FUNCTION_BLOCK FB_Station IMPLEMENTS ITF_Observable
VAR
	//ITF_Observable
	_Observers : ARRAY[1..2] OF ITF_Observer;
	_data	   : INT;
	prevData   : int;
END_VAR

METHOD CyclicLogic : BOOL
VAR
	dataChanged : BOOL;
END_VAR
//Monitor for change in data
IF data <> prevData THEN
	dataChanged := TRUE;
	prevData	:= Data;
END_IF

IF dataChanged THEN
	notifyObserver();
END_IF
END_METHOD

PROPERTY Data : int
GET
Data := _data;
END_GET
SET
_data := Data;
END_SET
END_PROPERTY

METHOD notifyObserver : BOOL
VAR
	i : UDINT;
END_VAR
FOR i := 1 TO 2 DO
	IF _Observers[i] <> 0 THEN
		_Observers[i].update(THIS^); //Call the update method of the observer and pass a reference to the Observable
	END_IF
END_FOR
END_METHOD

METHOD registerObserver : BOOL
VAR_INPUT
	Observer : ITF_Observer;
END_VAR

VAR
	i : UDINT;
END_VAR
//Find the first available array location and store a reference to the Observer there
FOR i := 1 TO 2 DO
	IF _Observers[i] = 0 THEN
		_Observers[i] := Observer;
		Observer.ID	  := i; //Send the location within the array back to the Observer, so it can pass the ID back when removing itself
		EXIT;
	END_IF
END_FOR
END_METHOD

METHOD removeObserver : BOOL
VAR_INPUT
	Observer : ITF_Observer;
END_VAR
//Check for valid reference
IF Observer <> 0 AND _Observers[Observer.ID] <> 0 THEN
	_Observers[Observer.ID] := 0; //Clear the array position
	Observer.ID				:= 0; //send back a 0 so the Observer knows it is no longer Observing
END_IF
END_METHOD

END_FUNCTION_BLOCK

(* stored: Version 1.1.0.1, ProductVersion 3.1.4024.12
   POU FB_Station: Id {4cffd1f8-e639-4cf1-8a94-e4412d1f6cef}, SpecialFunc None
   Folder ITF_Observable: Id {9faa726e-db41-4250-8f83-4ccb89e66920}
   Method CyclicLogic: Id {cf9a7094-bb19-4360-84cc-e74e74e0a599}
   Property Data: Id {137e3308-f419-4042-ae43-8222a8c628ab}
   Get Get: Id {63e77196-2361-45b1-8016-9b1810594e3b}
   Set Set: Id {73859c97-6c63-4604-94d8-4981cf36c3d5}
   Method notifyObserver: Id {5d01aa5d-a9ba-4807-b8f3-63e54734db00}
   Method registerObserver: Id {91468315-02a6-45bd-8a0e-94aeb2586c3a}
   Method removeObserver: Id {a3e6cb8e-a898-47c8-849c-012e0d5d387d} *)
